RoboDK station: dr608.rdk

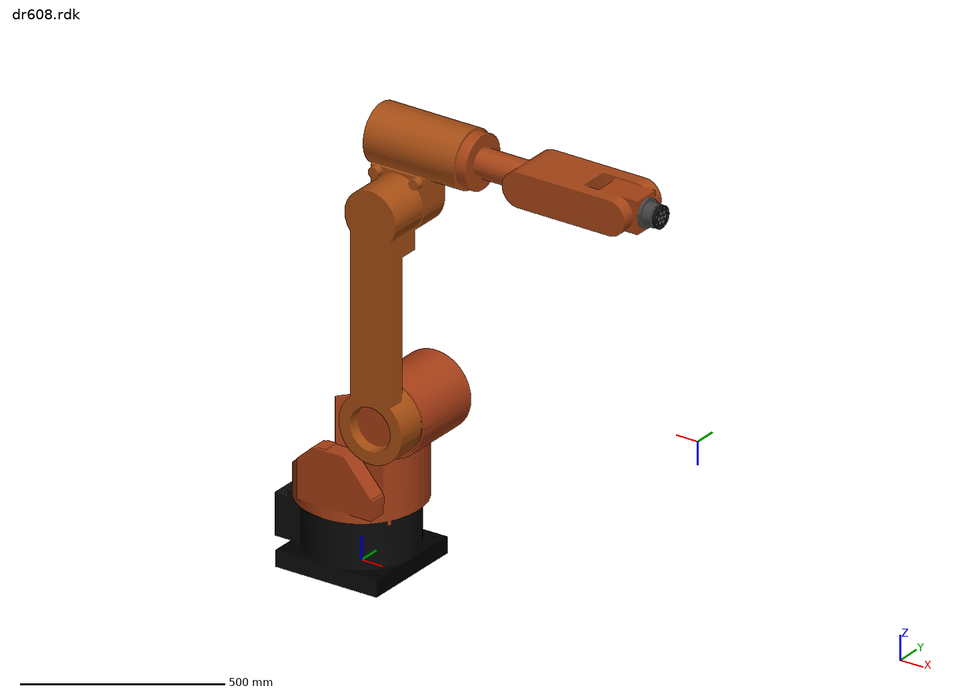
[picture v0: the station drawn from its stored meshes, robots at their saved joint values, targets as dots, program paths as lines]
Station dr608. Poses are relative to the parent item; angles as X-Y-Z fixed-axis rotations.
  - frame dr608 Base at (0, 0, 0) mm
    - robot dr608: 6 axes
        modified DH rows (alpha deg, a mm, theta deg, d mm): 0, 0, 0, 466; -90, 150, -90, 0; 0, 570, 0, 0; -90, 142.4, 0, 640; 90, 0, 0, 0; -90, 0, 180, 121.6
        joint limits [-180, -120, -130, -180, -115, -360] to [180, 120, 80, 180, 115, 360]; home [0, 0, 0, 0, 0, 0]; saved at [0, 0, 0, 0, 0, 0]
      - tool Tool 2, TCP at (0, 0, 0) mm
      - tool Weld gun, TCP at (-4, 0, 371.3) mm, rotated rx 0 ry 45 rz 0 deg, size 299.9 x 60 x 318.3 mm
      - tool Tool 3, TCP at (10, 10, 100) mm
    - frame Frame 2 at (1000, 0, 600) mm, rotated rx 180 ry 0 rz 180 deg
